(* PLC project Mixer, Sinergi Wahana Gemilang Unnamed 1, author Andi Sama *)
(* stored: creationDateTime 2022-08-10T22:53:50, companyURL www.swgemilang.com, modificationDateTime 2022-08-15T13:40:24 *)

PROGRAM Mixer
  VAR
    START AT %I0.0 : BOOL := FALSE;
    STOP AT %I0.1 : BOOL := FALSE;
    L_LEVEL AT %I0.2 : BOOL := FALSE;
    H_LEVEL AT %I0.3 : BOOL := FALSE;
    PUMP_1 AT %Q1.0 : BOOL := FALSE;
    PUMP_2 AT %Q2.0 : BOOL := FALSE;
    MIXER_MOTOR AT %Q3.0 : BOOL := FALSE;
  END_VAR
  VAR
    PT_MIXER_MOTOR : UINT := 10;
    SR0 : SR;
  END_VAR
  VAR
    VALVE AT %Q3.0 : BOOL := FALSE;
  END_VAR
  VAR
    SR1 : SR;
    ET_TON0 : TIME;
    TP0 : TP;
    F_TRIG0 : F_TRIG;
    RS0 : RS;
  END_VAR

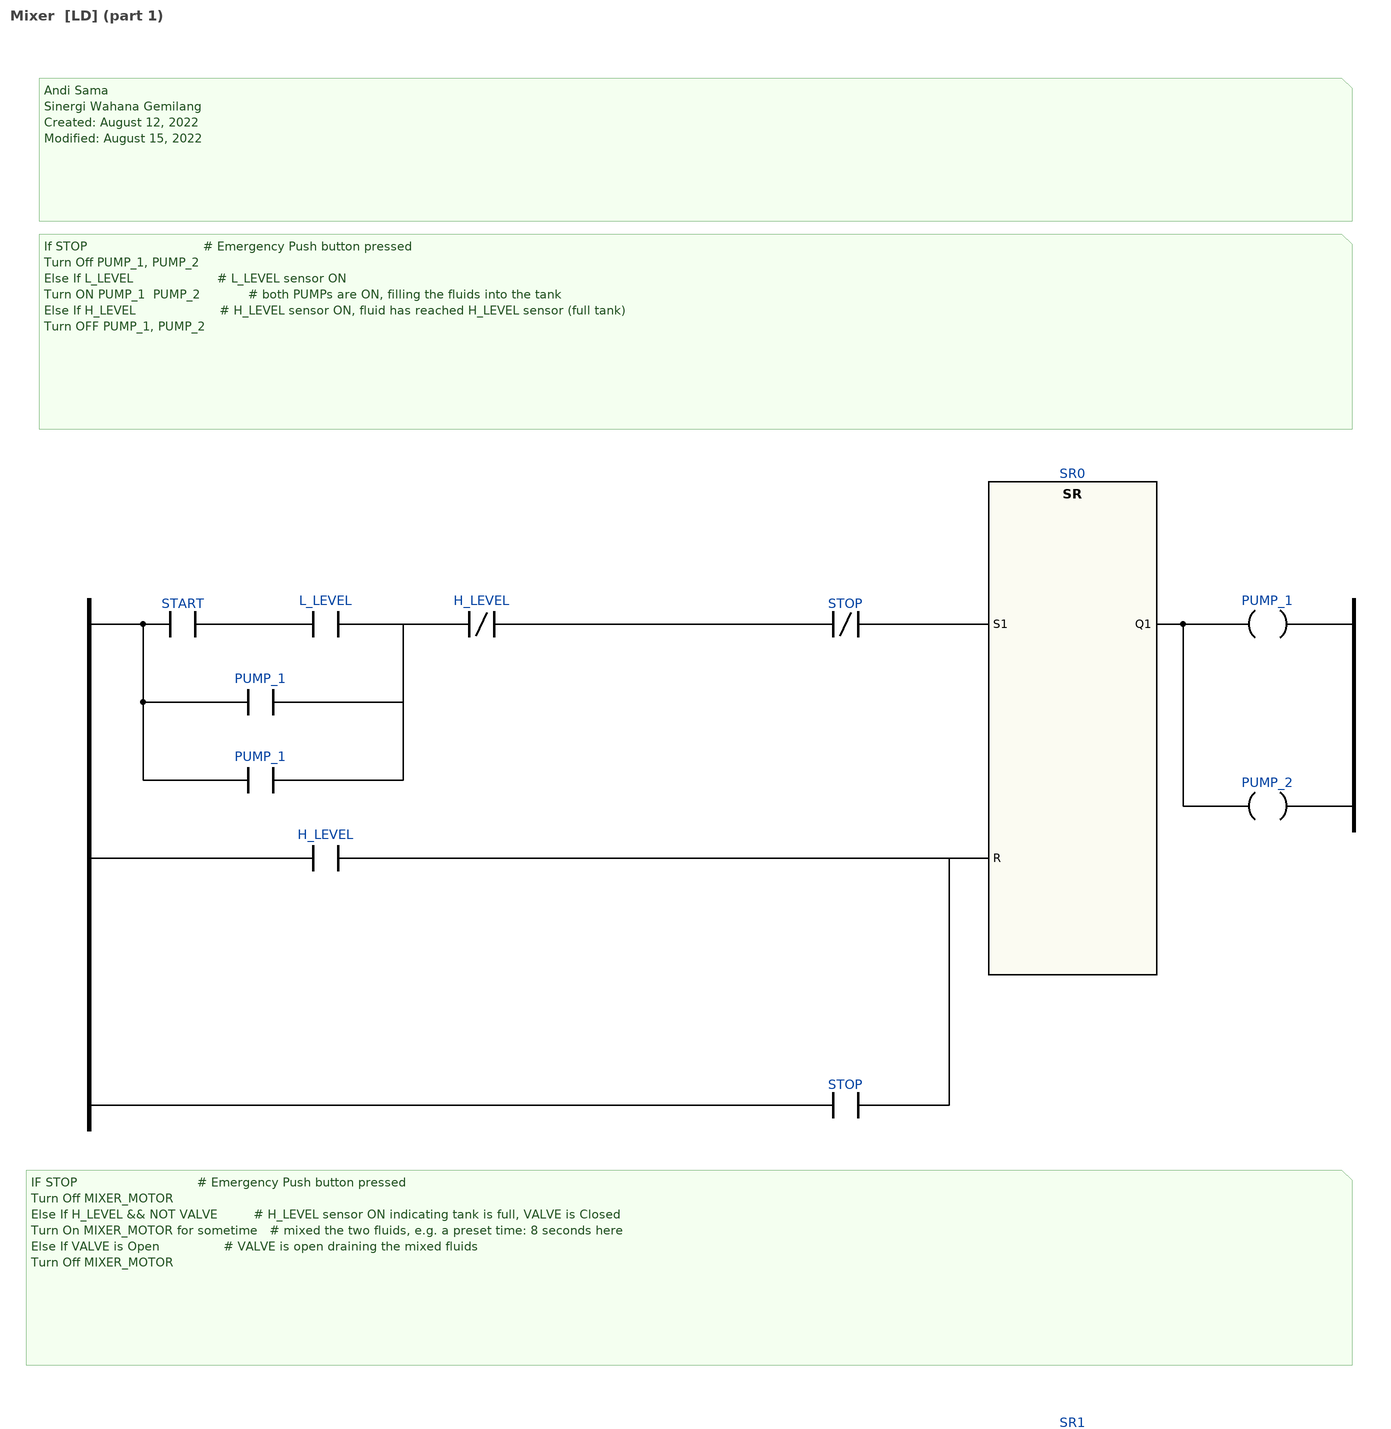
(* LD diagram, written out as Structured Text *)
(* Andi Sama
Sinergi Wahana Gemilang
Created: August 12, 2022
Modified: August 15, 2022 *)
(* If STOP                             # Emergency Push button pressed
  Turn Off PUMP_1, PUMP_2
Else If L_LEVEL                     # L_LEVEL sensor ON
  Turn ON PUMP_1  PUMP_2            # both PUMPs are ON, filling the fluids into the tank
Else If H_LEVEL                     # H_LEVEL sensor ON, fluid has reached H_LEVEL sensor (full tank)
  Turn OFF PUMP_1, PUMP_2 *)
SR0(S1 := (START AND L_LEVEL OR PUMP_1) AND NOT H_LEVEL AND NOT STOP, R := H_LEVEL OR STOP);
PUMP_1 := SR0.Q1;
PUMP_2 := SR0.Q1;
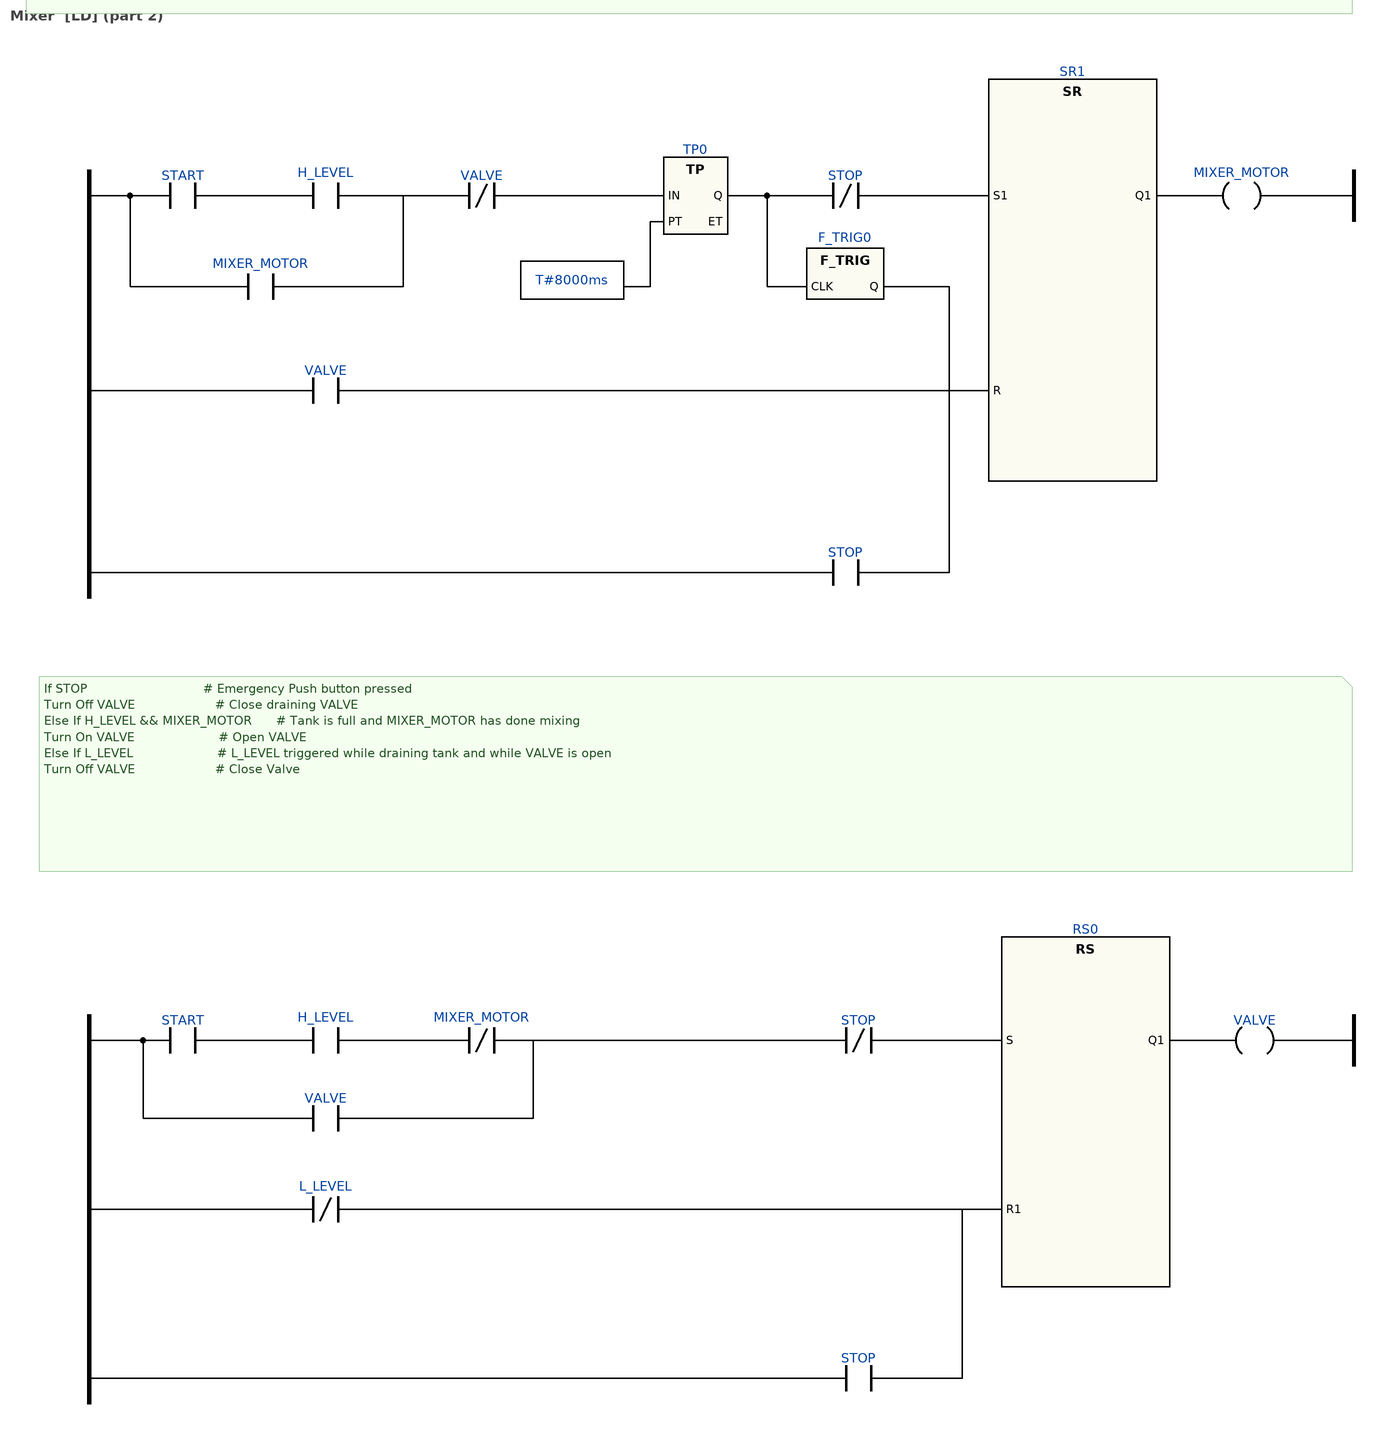
(* IF STOP                              # Emergency Push button pressed
  Turn Off MIXER_MOTOR 
Else If H_LEVEL && NOT VALVE         # H_LEVEL sensor ON indicating tank is full, VALVE is Closed
  Turn On MIXER_MOTOR for sometime   # mixed the two fluids, e.g. a preset time: 8 seconds here
Else If VALVE is Open                # VALVE is open draining the mixed fluids
  Turn Off MIXER_MOTOR *)
TP0(IN := (START AND H_LEVEL OR MIXER_MOTOR) AND NOT VALVE, PT := T#8000ms);
F_TRIG0(CLK := TP0.Q);
SR1(S1 := TP0.Q AND NOT STOP, R := STOP OR VALVE OR F_TRIG0.Q);
MIXER_MOTOR := SR1.Q1;
(* If STOP                             # Emergency Push button pressed
  Turn Off VALVE                    # Close draining VALVE
Else If H_LEVEL && MIXER_MOTOR      # Tank is full and MIXER_MOTOR has done mixing
  Turn On VALVE                     # Open VALVE
Else If L_LEVEL                     # L_LEVEL triggered while draining tank and while VALVE is open
  Turn Off VALVE                    # Close Valve *)
RS0(S := (START AND H_LEVEL AND NOT MIXER_MOTOR OR VALVE) AND NOT STOP, R1 := STOP OR NOT L_LEVEL);
VALVE := RS0.Q1;
END_PROGRAM

CONFIGURATION Config0
  RESOURCE Res0 ON PLC
    TASK task0(INTERVAL := T#20ms, PRIORITY := 0);
    PROGRAM instance0 WITH task0 : Mixer;
  END_RESOURCE
END_CONFIGURATION
